PROGRAM MAIN
VAR
	
	x: INT;
	y: INT;
	z: INT;
END_VAR

IF x > y THEN
	x := z;
ELSE
	x := x+1;
END_IF

END_PROGRAM

(* stored: Version 1.1.0.1, ProductVersion 3.1.4022.12
   POU MAIN: Id {c47f9aac-68c3-49c9-9898-0a3b0492dd80}, SpecialFunc None *)
